PROGRAM AutoStates_POU
VAR
END_VAR

END_PROGRAM

(* stored: Version 1.1.0.1, ProductVersion 3.1.4024.0
   POU AutoStates_POU: Id {56ee5f5c-2cf2-440e-8ce6-42e63b28d467}, SpecialFunc None *)
